{attribute 'qualified_only'}
VAR_GLOBAL
    stBasicMotor: DUT_MotionStage;
END_VAR

(* stored: Version 1.1.0.1, ProductVersion 3.1.4022.18
   GVL SIM: Id {93185b6e-16aa-4f8f-81ca-23800c58e227} *)
